{attribute 'qualified_only'}
{attribute 'strict'}
TYPE E_ActuatorCommand :
(
	Advance := 1,
	Retract := 2
);
END_TYPE

(* stored: Version 1.1.0.1, ProductVersion 3.1.4024.12
   DUT E_ActuatorCommand: Id {7b21bcdb-1032-4cba-85ee-663c80d42116} *)
